Omron CX-Programmer project 新工程 (CX-Programmer 9.73)

# PLC 新PLC1: CPM1(CPM1A) CPU30

## Program 新程序1 (no task)
; 这个PLC程序实现了一个称重系统的控制系统。 / 系统包含启动按钮、停止按钮、急停按钮、手动/自动开关、称重传感器信号、配料阀门开到位、配料阀门关到位、重量超限信号。 / 执行器包括配料阀门控制、显示器控制、报警灯、运行指示灯。 / 系统配备启动按钮用于启动，停止按钮用于正常停止，急停按钮用于紧急停止，手动/自动开关用于选择运行模式。 / 手动/自动开关设为自动时启用自动模式，否则启用手动模式。 / 在自动模式下，按下启动按钮后，若停止按钮未按下，系统置位系统运行标志，随后立即启动显示器控制显示称重数据，确保操作员能实时监控物料重量。 / 当启动按钮被按下，手动/自动开关设为自动，停止按钮未按下，称重传感器信号未检测到重量达到设定值，故障标志未置位且配料超时定时器未超时，系统置位配料阀门控制打开配料阀门，开始向容器中加入物料。 / 配料阀门控制在自动模式下且系统运行标志置位时打开，确保操作规范。当称重传感器信号检测到重量达到设定值时，配料阀门控制立即关闭，避免过量配料。 / 若生产过程中重量超限信号触发，表明物料重量超出安全范围，系统点亮报警灯，但需经过报警延时定时器的10个时间单位确认超限状态持续存在才会触发报警，以避免误报。当称重传感器信号或重量超限信号触发时，系统停止配料阀门控制，以保护设备安全。 / 若配料超时定时器超时，表明配料过程耗时过长，系统停止配料阀门控制，便于操作员检查设备。 / 在手动模式下，操作员通过手动配料按钮触发相关操作，实现灵活调整。 / 系统运行时，运行指示灯在进料阶段标志、搅拌阶段标志、出料阶段标志、维护阶段标志或故障标志任一置位时点亮，且通过运行指示灯延时定时器和运行指示灯熄灭延时定时器控制其闪烁时间，提供直观的状态反馈。

### Section 段1

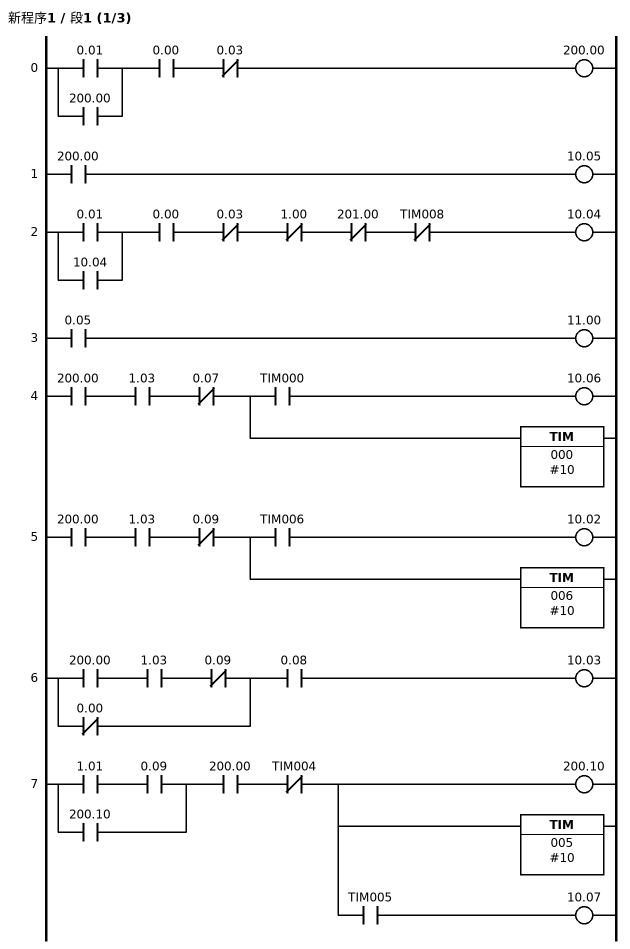
; rung 0
LD 0.01
OR 200.00
AND 0.00
ANDNOT 0.03
OUT 200.00
; rung 1
LD 200.00
OUT 10.05
; rung 2
LD 0.01
OR 10.04
AND 0.00
ANDNOT 0.03
ANDNOT 1.00
ANDNOT 201.00
ANDNOT TIM008
OUT 10.04
; rung 3
LD 0.05
OUT 11.00
; rung 4
LD 200.00
AND 1.03
ANDNOT 0.07
OUT TR0
AND TIM000
OUT 10.06
LD TR0
TIM 000 #10
; rung 5
LD 200.00
AND 1.03
ANDNOT 0.09
OUT TR0
AND TIM006
OUT 10.02
LD TR0
TIM 006 #10
; rung 6
LD 200.00
AND 1.03
ANDNOT 0.09
ORNOT 0.00
AND 0.08
OUT 10.03
; rung 7
LD 1.01
AND 0.09
OR 200.10
AND 200.00
ANDNOT TIM004
OUT 200.10
TIM 005 #10
AND TIM005
OUT 10.07

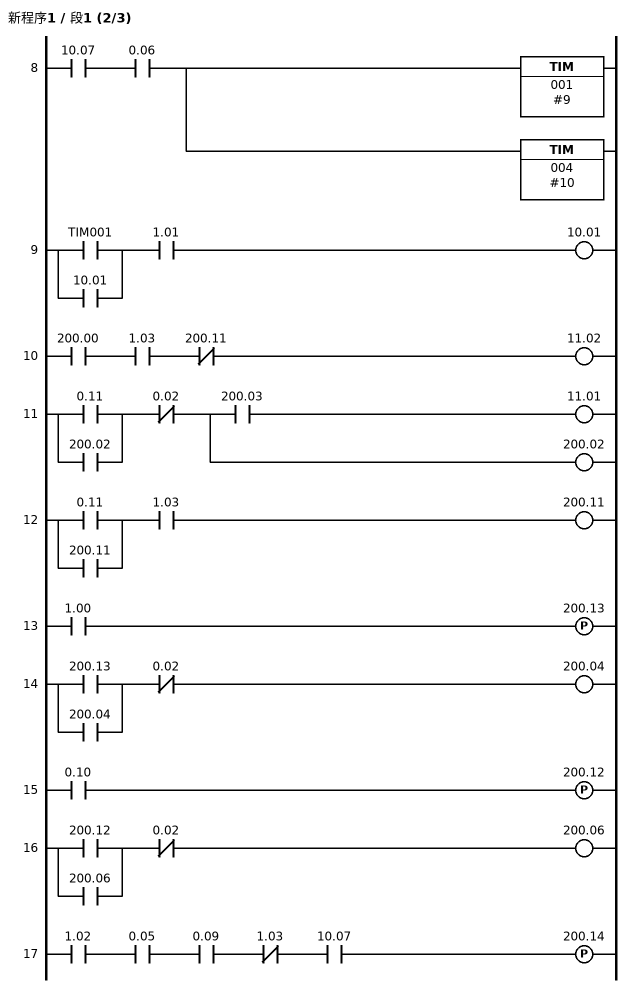
; rung 8
LD 10.07
AND 0.06
TIM 001 #9
TIM 004 #10
; rung 9
LD TIM001
OR 10.01
AND 1.01
OUT 10.01
; rung 10
LD 200.00
AND 1.03
ANDNOT 200.11
OUT 11.02
; rung 11
LD 0.11
OR 200.02
ANDNOT 0.02
OUT TR0
AND 200.03
OUT 11.01
LD TR0
OUT 200.02
; rung 12
LD 0.11
OR 200.11
AND 1.03
OUT 200.11
; rung 13
LD 1.00
DIFU(13) 200.13
; rung 14
LD 200.13
OR 200.04
ANDNOT 0.02
OUT 200.04
; rung 15
LD 0.10
DIFU(13) 200.12
; rung 16
LD 200.12
OR 200.06
ANDNOT 0.02
OUT 200.06
; rung 17
LD 1.02
AND 0.05
LD 0.09
ANDNOT 1.03
AND 10.07
ANDLD
DIFU(13) 200.14

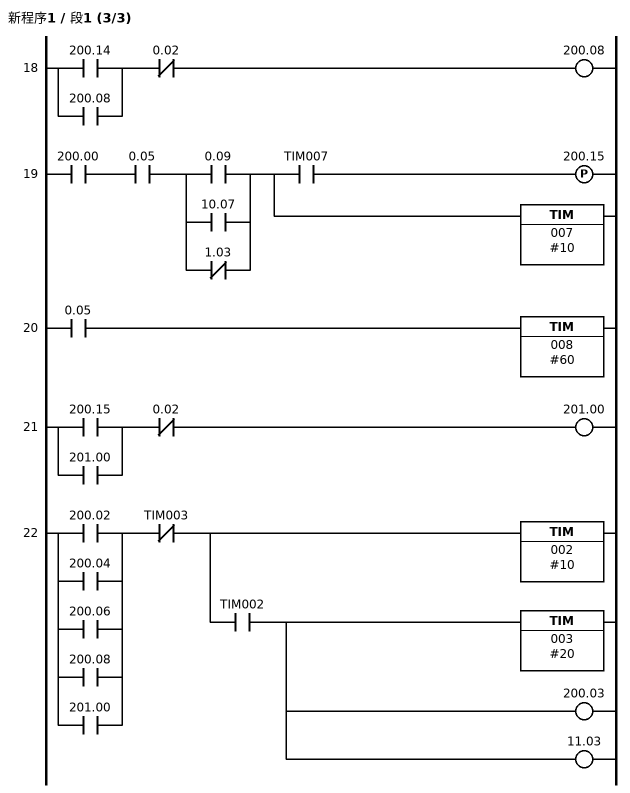
; rung 18
LD 200.14
OR 200.08
ANDNOT 0.02
OUT 200.08
; rung 19
LD 200.00
AND 0.05
LD 0.09
OR 10.07
ORNOT 1.03
ANDLD
OUT TR0
AND TIM007
DIFU(13) 200.15
LD TR0
TIM 007 #10
; rung 20
LD 0.05
TIM 008 #60
; rung 21
LD 200.15
OR 201.00
ANDNOT 0.02
OUT 201.00
; rung 22
LD 200.02
OR 200.04
OR 200.06
OR 200.08
OR 201.00
ANDNOT TIM003
TIM 002 #10
AND TIM002
TIM 003 #20
OUT 200.03
OUT 11.03
; rung 23
END(01)